(* CODESYS project Test ST.project

Project tree, tasks and I/O mapping:
  Device : CODESYS Control Win V3, 3S - Smart Software Solutions GmbH, version 3.5.15.30
    application Application
      libraries: Standard, * (System)
      task MainTask (cyclic, interval t#20ms, priority 1) calls PLC_PRG
      task VISU_TASK (cyclic, interval 100 ms, priority 31) calls VisuElems.Visu_Prg
      program PLC_PRG [ST]
      visualisation Visualization
  text list GlobalTextList
*)

// Device/Application/PLC_PRG
PROGRAM PLC_PRG
VAR
	Contact1 : BOOL := FALSE;
	Coil1 : BOOL;
END_VAR

IF Contact1 = TRUE THEN;
	Coil1 := TRUE;
ELSE
	Coil1 := FALSE;
END_IF

END_PROGRAM

// Device/Application/Visualization
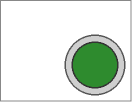
VISUALIZATION Visualization  // 132x102
    Lamp1 (60,30 70x70), variable: PLC_PRG.Coil1, style: Lamp-Lamp1-Green
END_VISUALIZATION
